PROGRAM PIST_CYCLE
VAR
	bFirstRun:BOOL:=FALSE;
	counter :INT;
END_VAR


grp_feeder();
grp_separate1();
grp_separate2();

ACTION grp_feeder:
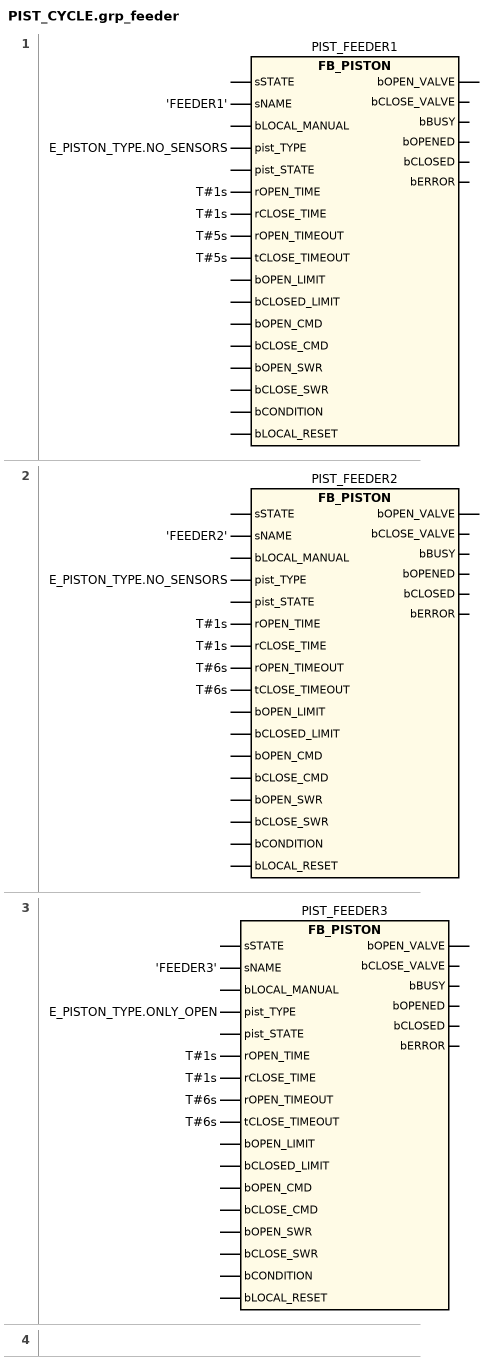
// NETWORK 1
PIST_FEEDER1(
    sNAME := 'FEEDER1',
    pist_TYPE := E_PISTON_TYPE.NO_SENSORS,
    rOPEN_TIME := T#1s,
    rCLOSE_TIME := T#1s,
    rOPEN_TIMEOUT := T#5s,
    tCLOSE_TIMEOUT := T#5s); // FB_PISTON

// NETWORK 2
PIST_FEEDER2(
    sNAME := 'FEEDER2',
    pist_TYPE := E_PISTON_TYPE.NO_SENSORS,
    rOPEN_TIME := T#1s,
    rCLOSE_TIME := T#1s,
    rOPEN_TIMEOUT := T#6s,
    tCLOSE_TIMEOUT := T#6s); // FB_PISTON

// NETWORK 3
PIST_FEEDER3(
    sNAME := 'FEEDER3',
    pist_TYPE := E_PISTON_TYPE.ONLY_OPEN,
    rOPEN_TIME := T#1s,
    rCLOSE_TIME := T#1s,
    rOPEN_TIMEOUT := T#6s,
    tCLOSE_TIMEOUT := T#6s); // FB_PISTON

// NETWORK 4
END_ACTION

ACTION grp_separate1:
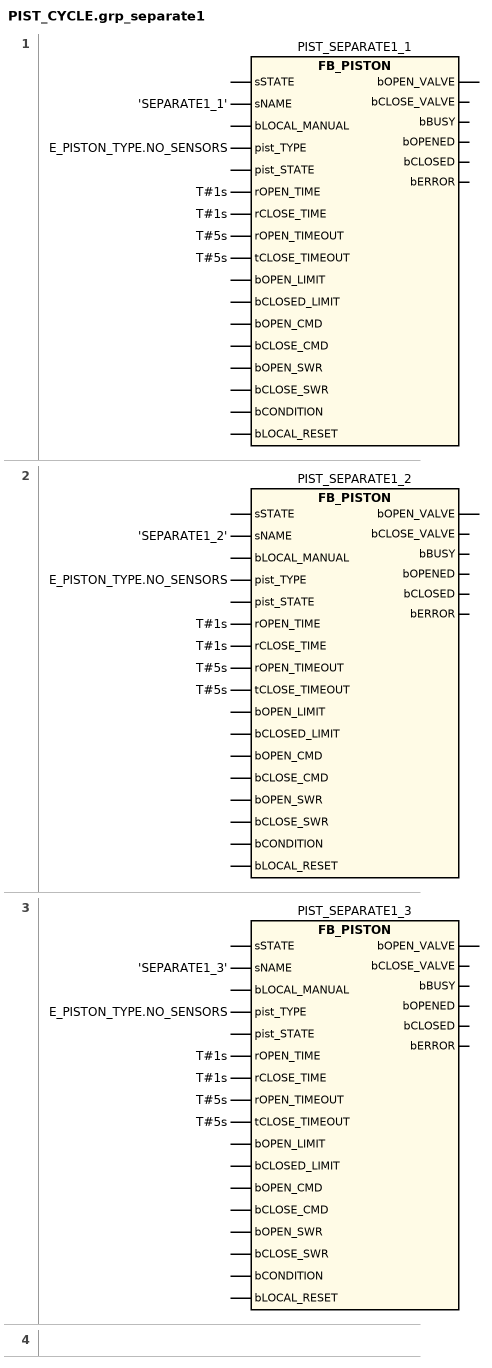
// NETWORK 1
PIST_SEPARATE1_1(
    sNAME := 'SEPARATE1_1',
    pist_TYPE := E_PISTON_TYPE.NO_SENSORS,
    rOPEN_TIME := T#1s,
    rCLOSE_TIME := T#1s,
    rOPEN_TIMEOUT := T#5s,
    tCLOSE_TIMEOUT := T#5s); // FB_PISTON

// NETWORK 2
PIST_SEPARATE1_2(
    sNAME := 'SEPARATE1_2',
    pist_TYPE := E_PISTON_TYPE.NO_SENSORS,
    rOPEN_TIME := T#1s,
    rCLOSE_TIME := T#1s,
    rOPEN_TIMEOUT := T#5s,
    tCLOSE_TIMEOUT := T#5s); // FB_PISTON

// NETWORK 3
PIST_SEPARATE1_3(
    sNAME := 'SEPARATE1_3',
    pist_TYPE := E_PISTON_TYPE.NO_SENSORS,
    rOPEN_TIME := T#1s,
    rCLOSE_TIME := T#1s,
    rOPEN_TIMEOUT := T#5s,
    tCLOSE_TIMEOUT := T#5s); // FB_PISTON

// NETWORK 4
END_ACTION

ACTION grp_separate2:
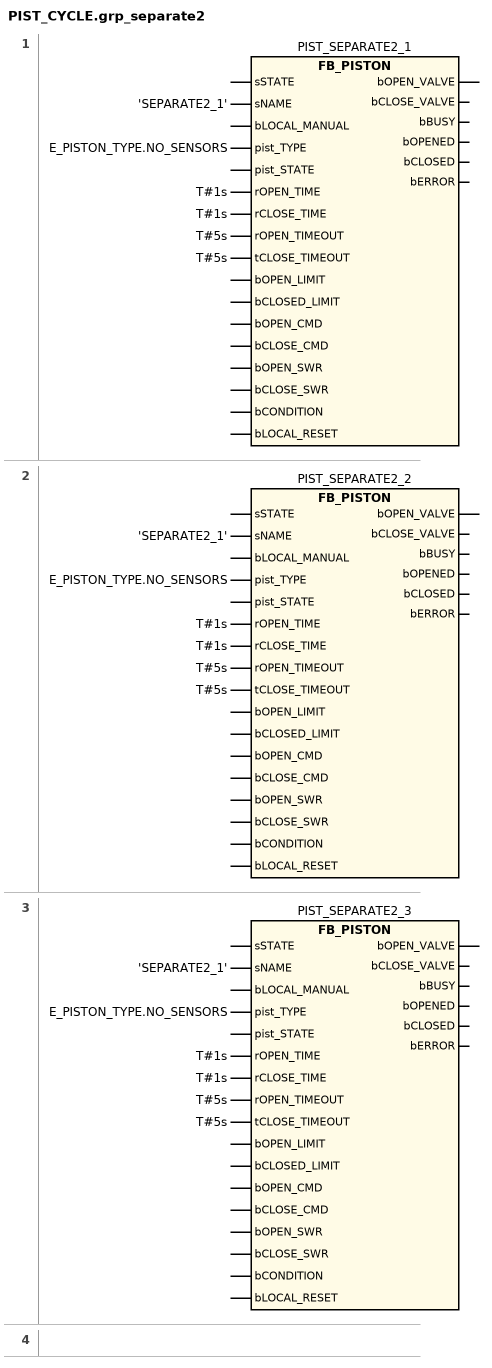
// NETWORK 1
PIST_SEPARATE2_1(
    sNAME := 'SEPARATE2_1',
    pist_TYPE := E_PISTON_TYPE.NO_SENSORS,
    rOPEN_TIME := T#1s,
    rCLOSE_TIME := T#1s,
    rOPEN_TIMEOUT := T#5s,
    tCLOSE_TIMEOUT := T#5s); // FB_PISTON

// NETWORK 2
PIST_SEPARATE2_2(
    sNAME := 'SEPARATE2_1',
    pist_TYPE := E_PISTON_TYPE.NO_SENSORS,
    rOPEN_TIME := T#1s,
    rCLOSE_TIME := T#1s,
    rOPEN_TIMEOUT := T#5s,
    tCLOSE_TIMEOUT := T#5s); // FB_PISTON

// NETWORK 3
PIST_SEPARATE2_3(
    sNAME := 'SEPARATE2_1',
    pist_TYPE := E_PISTON_TYPE.NO_SENSORS,
    rOPEN_TIME := T#1s,
    rCLOSE_TIME := T#1s,
    rOPEN_TIMEOUT := T#5s,
    tCLOSE_TIMEOUT := T#5s); // FB_PISTON

// NETWORK 4
END_ACTION

END_PROGRAM

(* stored: Version 1.1.0.1, ProductVersion 3.1.4024.12
   POU PIST_CYCLE: Id {b09e4efb-d7ec-45c6-bc50-8222237b347f}, SpecialFunc None
   Action grp_feeder: Id {b6db8f46-a5cd-4841-b2f4-af5cb236d344}
   Action grp_separate1: Id {c5a0a712-4fac-4232-a98c-d42134a9bfbf}
   Action grp_separate2: Id {1be0883d-7762-43b3-a9f8-21af8da01190} *)
